FUNCTION_BLOCK PUBLIC FB_Socket
VAR_OUTPUT
	bActive		: BOOL;
END_VAR

PROPERTY PUBLIC Active : BOOL
GET
Active := bActive;
END_GET
END_PROPERTY

METHOD PUBLIC Off
bActive := false;
END_METHOD

METHOD PUBLIC On
bActive := true;
END_METHOD

END_FUNCTION_BLOCK

(* stored: Version 1.1.0.1, ProductVersion 3.1.4020.3
   POU FB_Socket: Id {55e66dc1-05c3-43f8-9bc8-5075ca0cd865}, SpecialFunc None
   Property Active: Id {d6e4d23d-1261-40c6-80cc-51499451df21}
   Get Get: Id {3d5be9c4-7b0b-4454-a774-7d6c3fc8b550}
   Method Off: Id {54f23483-66d0-4707-9581-54558ff84187}
   Method On: Id {ea9cd1d9-8590-4b0b-b6ec-c19fb0ca1b1d} *)
